FUNCTION_BLOCK FB_Component_TE1 EXTENDS FB_BaseComponent IMPLEMENTS ITF_Component_TE1, ITF_Component_TE1_HMI_Init
VAR
END_VAR

METHOD testMethod : BOOL
VAR_INPUT
END_VAR
END_METHOD

END_FUNCTION_BLOCK

(* stored: Version 1.1.0.1, ProductVersion 3.1.4024.15
   POU FB_Component_TE1: Id {646a958d-e506-4710-b24c-19c523eda77a}, SpecialFunc None
   Method testMethod: Id {6bda535d-acc9-4b7d-bdbe-a365bae94f05} *)
